(*
  States for FB_FanucCycleStop.
  Sequence: Idle → Pulsing → Done (→ Idle)  [Standard mode]
            Idle → Pulsing → WaitStop → Done (→ Idle)  [Abort mode]
  Error on timeout in WaitStop; reset by setting bTrigger FALSE.
*)
TYPE E_FanucCstopiState :
(
	Idle     := 0,   // Waiting for bTrigger rising edge.
	Pulsing  := 1,   // CSTOPI signal pulsed for 20 ms.
	WaitStop := 2,   // Abort mode only: waiting for bPrg_Running = FALSE (timeout → Error).
	Done     := 3,   // Cycle stop complete – bDone TRUE for one scan, then → Idle.
	Error    := 99   // Abort mode: program did not stop in time. Set bTrigger FALSE to reset.
);
END_TYPE

(* stored: Version 1.1.0.1, ProductVersion 3.1.4026.18
   DUT E_FanucCstopiState: Id {c3d4e5f6-a7b8-9012-cdef-012345678902} *)
